{attribute addProperty BoxType "EL5102-0000-0016"}
{attribute addProperty Id "StatusAT %I*Status_A99988373241Counter_valueAT %I*UDINT32417Latch_valueAT %I*UDINT32418Latch_value_2AT %I*UDINT32434"}
{attribute addProperty CRC "3618286503"}
{attribute addProperty SizeInBites "128"}
{attribute addProperty SizeInBytes "16"}
TYPE ENC_Status_Channel_D7AAABA7 :
STRUCT
	{attribute addProperty Name "Status"}
	Status AT %I* : Status_A9998837;
	{attribute addProperty Name "Counter_value"}
	Counter_value AT %I* : UDINT;
	{attribute addProperty Name "Latch_value"}
	Latch_value AT %I* : UDINT;
	{attribute addProperty Name "Latch_value_2"}
	Latch_value_2 AT %I* : UDINT;
END_STRUCT
END_TYPE

(* stored: Version 1.2.0.0, ProductVersion 3.1.4024.9
   DUT ENC_Status_Channel_D7AAABA7: Id {415bca58-e302-4ba4-bd48-5782666cfd58} *)
